{attribute addProperty BoxType "IODEVICETYPE_ETHERCATPROT"}
{attribute addProperty Id "Beckhoff_EK11xxBeckhoff_EK11xx_C12453FF49061.25Beckhoff_EK12xxBeckhoff_EK12xx_26FD3E4A162Beckhoff_EK13xxBeckhoff_EK13xx_F78FC0F811814.75Beckhoff_EK15xxBeckhoff_EK15xx_2CCE234B61476.75Beckhoff_EK18xxBeckhoff_EK18xx_2BB313921271158.875Beckhoff_EKM1xxxBeckhoff_EKM1xxx_A6D532072586323.25Beckhoff_EKx9xxBeckhoff_EKx9xx_143049714464558Beckhoff_EKxxxx_0080Beckhoff_EKxxxx_0080_F8E2E0BC648SyncUnitsSyncUnits_BBFB8ED413016.25InputsInputs_C3133F881088136OutputsOutputs_BAAAC74672090InfoDataInfoData_E9F65A829612"}
{attribute addProperty CRC "183930965"}
{attribute addProperty SizeInBites "11657"}
{attribute addProperty SizeInBytes "1457.125"}
TYPE EtherCAT_Master_EKxxxx_0AF69055 :
STRUCT
	{attribute addProperty Name "Beckhoff_EK11xx"}
	Beckhoff_EK11xx : Beckhoff_EK11xx_C12453FF;
	{attribute addProperty Name "Beckhoff_EK12xx"}
	Beckhoff_EK12xx : Beckhoff_EK12xx_26FD3E4A;
	{attribute addProperty Name "Beckhoff_EK13xx"}
	Beckhoff_EK13xx : Beckhoff_EK13xx_F78FC0F8;
	{attribute addProperty Name "Beckhoff_EK15xx"}
	Beckhoff_EK15xx : Beckhoff_EK15xx_2CCE234B;
	{attribute addProperty Name "Beckhoff_EK18xx"}
	Beckhoff_EK18xx : Beckhoff_EK18xx_2BB31392;
	{attribute addProperty Name "Beckhoff_EKM1xxx"}
	Beckhoff_EKM1xxx : Beckhoff_EKM1xxx_A6D53207;
	{attribute addProperty Name "Beckhoff_EKx9xx"}
	Beckhoff_EKx9xx : Beckhoff_EKx9xx_14304971;
	{attribute addProperty Name "Beckhoff_EKxxxx_0080"}
	Beckhoff_EKxxxx_0080 : Beckhoff_EKxxxx_0080_F8E2E0BC;
	{attribute addProperty Name "SyncUnits"}
	SyncUnits : SyncUnits_BBFB8ED4;
	{attribute addProperty Name "Inputs"}
	Inputs : Inputs_C3133F88;
	{attribute addProperty Name "Outputs"}
	Outputs : Outputs_BAAAC746;
	{attribute addProperty Name "InfoData"}
	InfoData : InfoData_E9F65A82;
END_STRUCT
END_TYPE

(* stored: Version 1.2.0.0, ProductVersion 3.1.4024.9
   DUT EtherCAT_Master_EKxxxx_0AF69055: Id {f607fce6-3a48-4705-8333-c1ccc3852e15} *)
